FUNCTION_BLOCK RunPnueIndexer EXTENDS RunUnitIndexerMaster
VAR_INPUT
END_VAR
VAR_OUTPUT
END_VAR
VAR
	//devices
	lockCylinder : POINTER TO RunCylinder;
	pistonCylinder : POINTER TO RunCylinder;
	
	sensorPairs : ARRAY[0..3] OF defSensorPair; //define stations sensor flag signatures
	fixtures : POINTER TO helperOutputSelection;
	
	//----------------
	//	Initialization
	//----------------
	revolveCounter : INT;
	revolveGoal : INT;
END_VAR

SUPER^(); //run indexer master

CASE outputState OF
	//---------------------------
	//	Initialization : revolve n times
	//---------------------------	
	eSpecialStates.INITIAL_BEGIN:
		revolveCounter:=0;
		bSerialTransition := TRUE;
	eSpecialStates.INITIAL_STATE_1:
		bSerialTransition := lockCylinder^.Execute(eCylinderCommands.COMMAND_B);
	eSpecialStates.INITIAL_STATE_2:
		bSerialTransition := pistonCylinder^.Execute(eCylinderCommands.COMMAND_B);
	eSpecialStates.INITIAL_STATE_3:
		bSerialTransition := lockCylinder^.Execute(eCylinderCommands.COMMAND_A);
	eSpecialStates.INITIAL_STATE_4:
		bSerialTransition := pistonCylinder^.Execute(eCylinderCommands.COMMAND_A);
		IF bSerialTransition THEN
			revolveCounter := revolveCounter+1;
			IF revolveCounter < revolveGoal THEN
				NextState := eSpecialStates.INITIAL_STATE_1; //repeat
			ELSE
				NextState := eSpecialStates.INITIAL_STATE_5; //to lock
			END_IF	
		END_IF
	eSpecialStates.INITIAL_STATE_5:
		bSerialTransition := lockCylinder^.Execute(eCylinderCommands.COMMAND_B);
		IF bSerialTransition THEN
			NextState := eSpecialStates.INITIAL_END; //terminated
		END_IF
	//------------------start running
	// S16#10 - : setup vacuum fixtures
	// S16#20 - : pnuematic indexer movement
	// 1. unlock
	// 2. shift out
	// 3. lock
	//------------------
	16#10:
		//activate fixture by slot valid status
		FOR nCounter := 0 TO SlotCount-1 BY 1 DO
			fixtures^.Trigger(sensorPairs[nCounter],SlotBase[nCounter].Valid); //TODO , not linked
		END_FOR
		NextState := 16#20;
	//----------
	16#20:
		bSerialTransition := pistonCylinder^.Execute(eCylinderCommands.COMMAND_B);
	16#21:
		bSerialTransition := lockCylinder^.Execute(eCylinderCommands.COMMAND_A);
	16#22:
		bSerialTransition := pistonCylinder^.Execute(eCylinderCommands.COMMAND_A);
	16#23:
		bSerialTransition := lockCylinder^.Execute(eCylinderCommands.COMMAND_B);
		IF bSerialTransition THEN
			fixtures^.ReleaseAll(); //release all fixture
			NextState := 16#0F; //join master sequence
		END_IF
END_CASE

METHOD FB_init : BOOL
VAR_INPUT
	bInitRetains : BOOL; // if TRUE, the retain variables are initialized (warm start / cold start)
	bInCopyCode : BOOL;  // if TRUE, the instance afterwards gets moved into the copy code (online change)
	
	argParent : POINTER TO RunUnitGeneric;
	argSlotBase : POINTER TO RunMaterial;
	argSlotLast : POINTER TO RunMaterial;
	
	argUpstream : POINTER TO RunUnitTransporterBase;
	argAxis : POINTER TO RunAxis;
	
	argLockCylinder : POINTER TO RunCylinder;
	argPistonCylinder : POINTER TO RunCylinder;
END_VAR
//initialize 
Parent := argParent;
SlotBase := argSlotBase;
SlotLast := argSlotLast;

Axis := argAxis;
Upstream := argUpstream;

isProxyMode:=FALSE; //no proxy


//calculate how much slot related
SlotCount :=  TO_INT((SlotLast-SlotBase)/SIZEOF(RunMaterial) + 1);

lockCylinder := argLockCylinder;
pistonCylinder := argPistonCylinder;
END_METHOD

END_FUNCTION_BLOCK

(* stored: Version 1.1.0.1, ProductVersion 3.1.4024.0
   POU RunPnueIndexer: Id {0282178a-e4a8-43e2-88ce-00a99b488386}, SpecialFunc None
   Method FB_init: Id {8dfee478-70bf-4472-a4ae-21e0c723276a} *)
